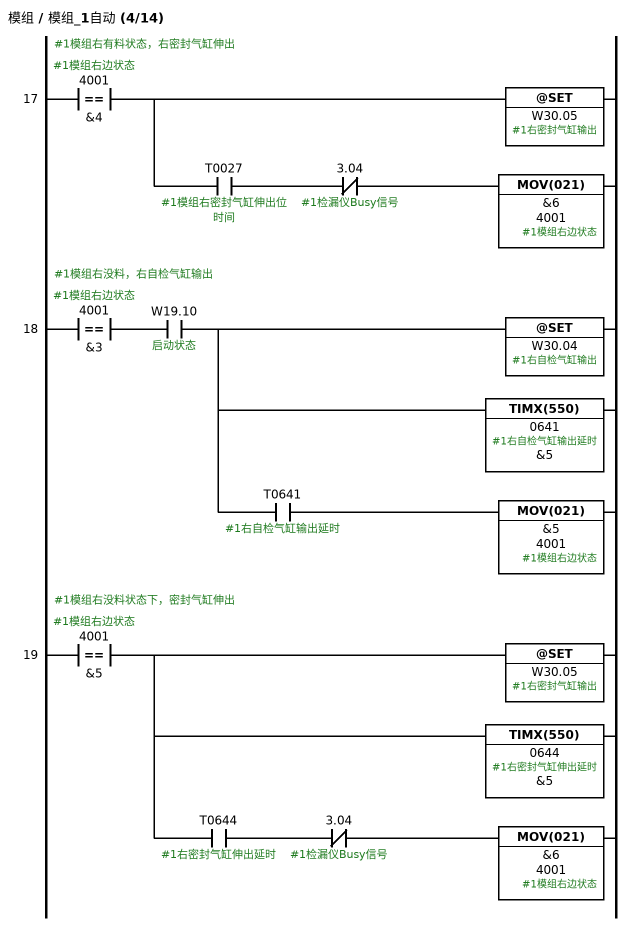
; [picture p209: 模组 / 模组_1自动, rungs 17-19]
; rung 17: #1模组右有料状态，右密封气缸伸出
LD=(300) 4001 &4  ; #1模组右边状态
@SET W30.05  ; #1右密封气缸输出
AND T0027  ; #1模组右密封气缸伸出位时间
ANDNOT 3.04  ; #1检漏仪Busy信号
MOV(021) &6 4001  ; #1模组右边状态
; rung 18: #1模组右没料，右自检气缸输出
LD=(300) 4001 &3  ; #1模组右边状态
AND W19.10  ; 启动状态
@SET W30.04  ; #1右自检气缸输出
TIMX(550) 0641 &5  ; #1右自检气缸输出延时
AND T0641  ; #1右自检气缸输出延时
MOV(021) &5 4001  ; #1模组右边状态
; rung 19: #1模组右没料状态下，密封气缸伸出
LD=(300) 4001 &5  ; #1模组右边状态
@SET W30.05  ; #1右密封气缸输出
TIMX(550) 0644 &5  ; #1右密封气缸伸出延时
AND T0644  ; #1右密封气缸伸出延时
ANDNOT 3.04  ; #1检漏仪Busy信号
MOV(021) &6 4001  ; #1模组右边状态

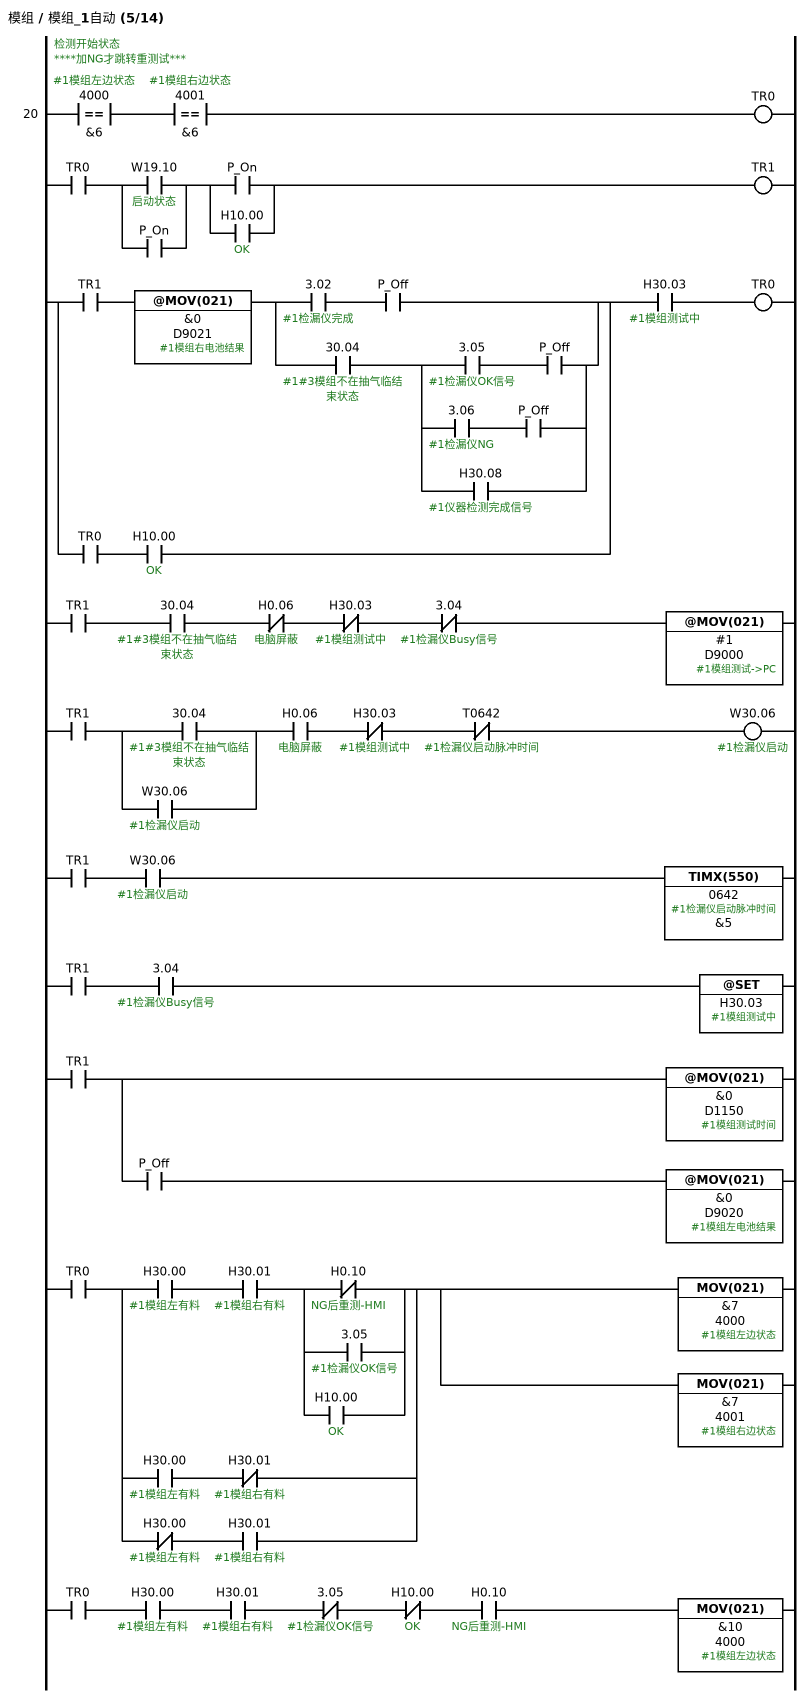
; rung 20: 检测开始状态 / ****加NG才跳转重测试***
LD=(300) 4000 &6  ; #1模组左边状态
AND=(300) 4001 &6  ; #1模组右边状态
OUT TR0
LD W19.10  ; 启动状态
OR P_On
ANDLD
LD P_On
OR H10.00  ; OK
ANDLD
OUT TR1
AND 30.04  ; #1#3模组不在抽气临结束状态  // 2018/5/28hy修改 所有模组不在抽气临结束状态下，下一模组才能启动(防抽气NG)
ANDNOT H0.06  ; 电脑屏蔽
ANDNOT H30.03  ; #1模组测试中
ANDNOT 3.04  ; #1检漏仪Busy信号
@MOV(021) #1 D9000  ; #1模组测试->PC
LD TR1
LD 30.04  ; #1#3模组不在抽气临结束状态  // 2018/5/28hy修改 所有模组不在抽气临结束状态下，下一模组才能启动(防抽气NG)
OR W30.06  ; #1检漏仪启动
ANDLD
AND H0.06  ; 电脑屏蔽
ANDNOT H30.03  ; #1模组测试中
ANDNOT T0642  ; #1检漏仪启动脉冲时间
OUT W30.06  ; #1检漏仪启动
LD TR1
AND W30.06  ; #1检漏仪启动
TIMX(550) 0642 &5  ; #1检漏仪启动脉冲时间
LD TR1
AND 3.04  ; #1检漏仪Busy信号
@SET H30.03  ; #1模组测试中
LD TR1
@MOV(021) &0 D1150  ; #1模组测试时间
AND P_Off
@MOV(021) &0 D9020  ; #1模组左电池结果
LD TR1
@MOV(021) &0 D9021  ; #1模组右电池结果
LD 3.02  ; #1检漏仪完成
AND P_Off
LD 30.04  ; #1#3模组不在抽气临结束状态  // 2018/5/29hy修改,所有模组不在临抽气结束状态下，测试模组测试完成后，给出停止测试信号
LD 3.05  ; #1检漏仪OK信号
AND P_Off
LD 3.06  ; #1检漏仪NG
AND P_Off
ORLD
OR H30.08  ; #1仪器检测完成信号
ANDLD
ORLD
ANDLD
LD TR0
AND H10.00  ; OK
ORLD
AND H30.03  ; #1模组测试中
OUT TR0
LD H30.00  ; #1模组左有料
AND H30.01  ; #1模组右有料
LDNOT H0.10  ; NG后重测-HMI
OR 3.05  ; #1检漏仪OK信号
OR H10.00  ; OK
ANDLD
LD H30.00  ; #1模组左有料
ANDNOT H30.01  ; #1模组右有料
ORLD
LDNOT H30.00  ; #1模组左有料
AND H30.01  ; #1模组右有料
ORLD
ANDLD
MOV(021) &7 4000  ; #1模组左边状态
MOV(021) &7 4001  ; #1模组右边状态
LD TR0
AND H30.00  ; #1模组左有料
AND H30.01  ; #1模组右有料
ANDNOT 3.05  ; #1检漏仪OK信号
ANDNOT H10.00  ; OK
AND H0.10  ; NG后重测-HMI
MOV(021) &10 4000  ; #1模组左边状态

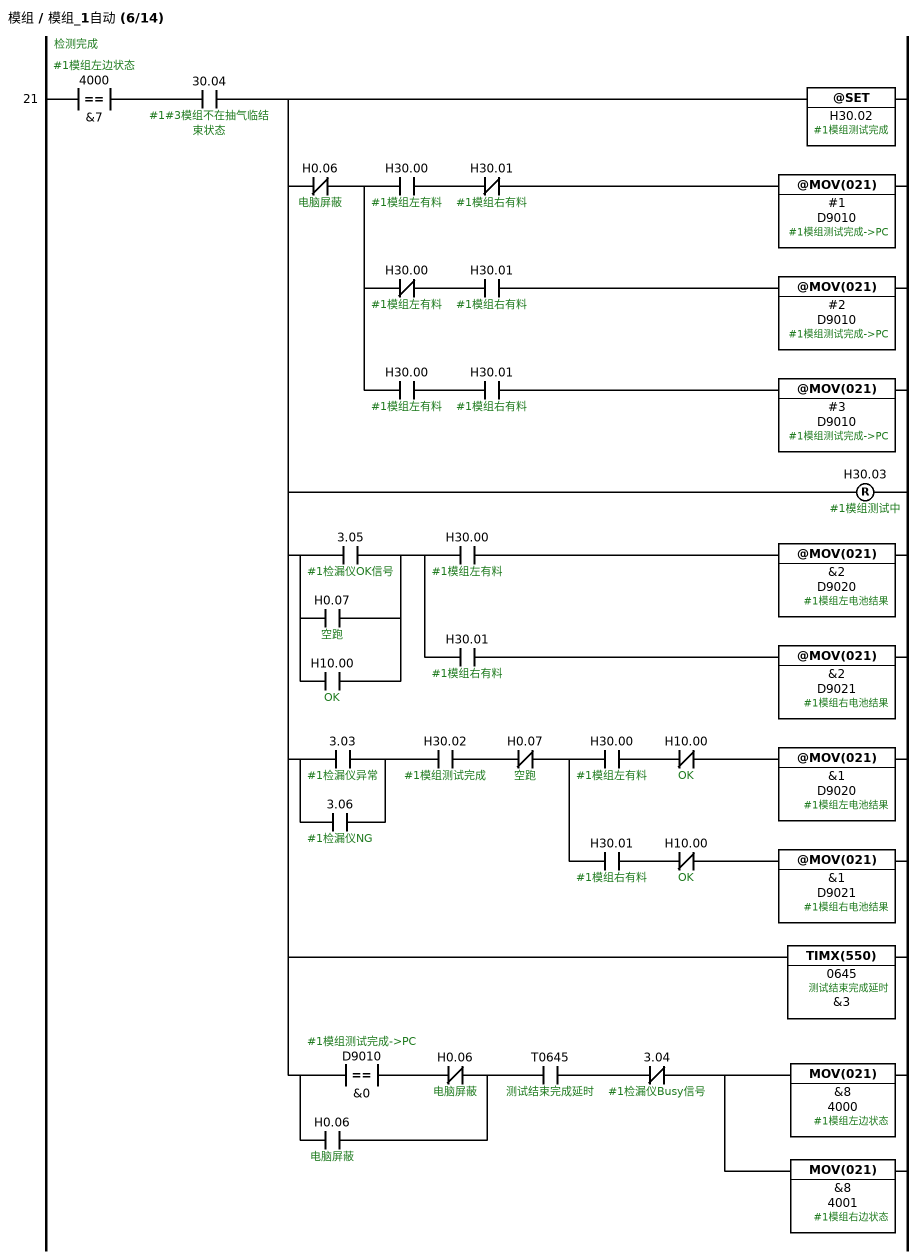
; rung 21: 检测完成
LD=(300) 4000 &7  ; #1模组左边状态
AND 30.04  ; #1#3模组不在抽气临结束状态
OUT TR0
@SET H30.02  ; #1模组测试完成
ANDNOT H0.06  ; 电脑屏蔽
OUT TR1
AND H30.00  ; #1模组左有料
ANDNOT H30.01  ; #1模组右有料
@MOV(021) #1 D9010  ; #1模组测试完成->PC
LD TR1
ANDNOT H30.00  ; #1模组左有料
AND H30.01  ; #1模组右有料
@MOV(021) #2 D9010  ; #1模组测试完成->PC
LD TR1
AND H30.00  ; #1模组左有料
AND H30.01  ; #1模组右有料
@MOV(021) #3 D9010  ; #1模组测试完成->PC
LD TR0
RSET H30.03  ; #1模组测试中
LD 3.05  ; #1检漏仪OK信号
OR H0.07  ; 空跑
OR H10.00  ; OK
ANDLD
OUT TR1
AND H30.00  ; #1模组左有料
@MOV(021) &2 D9020  ; #1模组左电池结果
LD TR1
AND H30.01  ; #1模组右有料
@MOV(021) &2 D9021  ; #1模组右电池结果
LD TR0
LD 3.03  ; #1检漏仪异常
OR 3.06  ; #1检漏仪NG
ANDLD
AND H30.02  ; #1模组测试完成
ANDNOT H0.07  ; 空跑
OUT TR1
AND H30.00  ; #1模组左有料
ANDNOT H10.00  ; OK
@MOV(021) &1 D9020  ; #1模组左电池结果
LD TR1
AND H30.01  ; #1模组右有料
ANDNOT H10.00  ; OK
@MOV(021) &1 D9021  ; #1模组右电池结果
LD TR0
TIMX(550) 0645 &3  ; 测试结束完成延时
LD=(300) D9010 &0  ; #1模组测试完成->PC
ANDNOT H0.06  ; 电脑屏蔽
OR H0.06  ; 电脑屏蔽
ANDLD
AND T0645  ; 测试结束完成延时
ANDNOT 3.04  ; #1检漏仪Busy信号
MOV(021) &8 4000  ; #1模组左边状态
MOV(021) &8 4001  ; #1模组右边状态

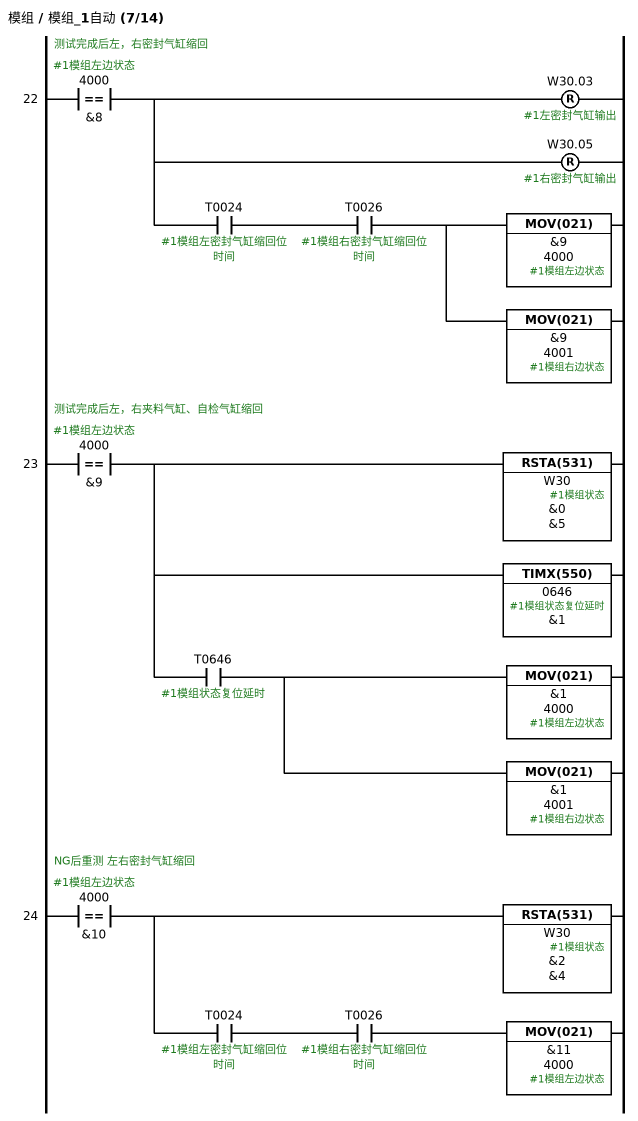
; rung 22: 测试完成后左，右密封气缸缩回
LD=(300) 4000 &8  ; #1模组左边状态
RSET W30.03  ; #1左密封气缸输出
RSET W30.05  ; #1右密封气缸输出
AND T0024  ; #1模组左密封气缸缩回位时间
AND T0026  ; #1模组右密封气缸缩回位时间
MOV(021) &9 4000  ; #1模组左边状态
MOV(021) &9 4001  ; #1模组右边状态
; rung 23: 测试完成后左，右夹料气缸、自检气缸缩回
LD=(300) 4000 &9  ; #1模组左边状态
RSTA(531) W30 &0 &5  ; #1模组状态
TIMX(550) 0646 &1  ; #1模组状态复位延时
AND T0646  ; #1模组状态复位延时
MOV(021) &1 4000  ; #1模组左边状态
MOV(021) &1 4001  ; #1模组右边状态
; rung 24: NG后重测 左右密封气缸缩回
LD=(300) 4000 &10  ; #1模组左边状态
RSTA(531) W30 &2 &4  ; #1模组状态
AND T0024  ; #1模组左密封气缸缩回位时间
AND T0026  ; #1模组右密封气缸缩回位时间
MOV(021) &11 4000  ; #1模组左边状态

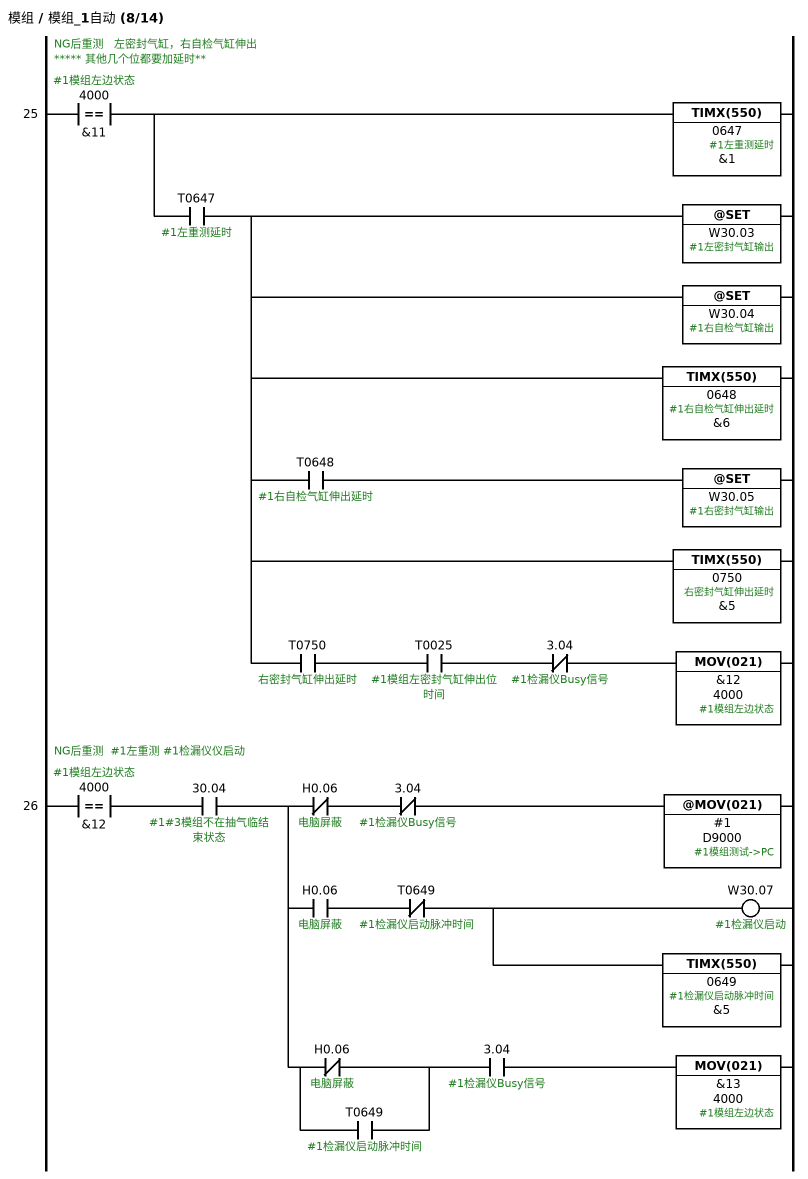
; rung 25: NG后重测   左密封气缸，右自检气缸伸出 / ***** 其他几个位都要加延时**
LD=(300) 4000 &11  ; #1模组左边状态
TIMX(550) 0647 &1  ; #1左重测延时
AND T0647  ; #1左重测延时
OUT TR0
@SET W30.03  ; #1左密封气缸输出
@SET W30.04  ; #1右自检气缸输出
TIMX(550) 0648 &6  ; #1右自检气缸伸出延时
AND T0648  ; #1右自检气缸伸出延时
@SET W30.05  ; #1右密封气缸输出
LD TR0
TIMX(550) 0750 &5  ; 右密封气缸伸出延时
AND T0750  ; 右密封气缸伸出延时
AND T0025  ; #1模组左密封气缸伸出位时间
ANDNOT 3.04  ; #1检漏仪Busy信号
MOV(021) &12 4000  ; #1模组左边状态
; rung 26: NG后重测  #1左重测 #1检漏仪仪启动
LD=(300) 4000 &12  ; #1模组左边状态
AND 30.04  ; #1#3模组不在抽气临结束状态  // 2018/5/28hy修改 所有模组不在抽气临结束状态下，下一模组才能启动(防抽气NG)
OUT TR0
ANDNOT H0.06  ; 电脑屏蔽
ANDNOT 3.04  ; #1检漏仪Busy信号
@MOV(021) #1 D9000  ; #1模组测试->PC
LD TR0
AND H0.06  ; 电脑屏蔽
ANDNOT T0649  ; #1检漏仪启动脉冲时间
OUT W30.07  ; #1检漏仪启动
TIMX(550) 0649 &5  ; #1检漏仪启动脉冲时间
LD TR0
LDNOT H0.06  ; 电脑屏蔽
OR T0649  ; #1检漏仪启动脉冲时间
ANDLD
AND 3.04  ; #1检漏仪Busy信号
MOV(021) &13 4000  ; #1模组左边状态

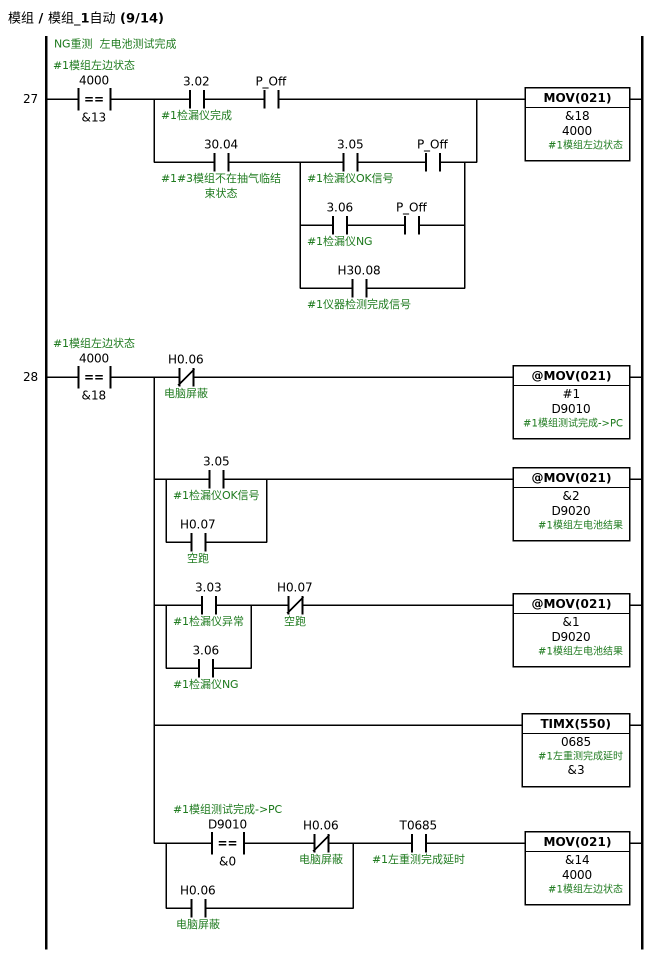
; rung 27: NG重测  左电池测试完成
LD=(300) 4000 &13  ; #1模组左边状态
LD 3.02  ; #1检漏仪完成
AND P_Off
LD 30.04  ; #1#3模组不在抽气临结束状态  // 2018/5/29hy修改,所有模组不在临抽气结束状态下，测试模组测试完成后，给出停止测试信号
LD 3.05  ; #1检漏仪OK信号
AND P_Off
LD 3.06  ; #1检漏仪NG
AND P_Off
ORLD
OR H30.08  ; #1仪器检测完成信号
ANDLD
ORLD
ANDLD
MOV(021) &18 4000  ; #1模组左边状态
; rung 28
LD=(300) 4000 &18  ; #1模组左边状态
OUT TR0
ANDNOT H0.06  ; 电脑屏蔽
@MOV(021) #1 D9010  ; #1模组测试完成->PC
LD TR0
LD 3.05  ; #1检漏仪OK信号
OR H0.07  ; 空跑
ANDLD
@MOV(021) &2 D9020  ; #1模组左电池结果
LD TR0
LD 3.03  ; #1检漏仪异常
OR 3.06  ; #1检漏仪NG
ANDLD
ANDNOT H0.07  ; 空跑
@MOV(021) &1 D9020  ; #1模组左电池结果
LD TR0
TIMX(550) 0685 &3  ; #1左重测完成延时
LD=(300) D9010 &0  ; #1模组测试完成->PC
ANDNOT H0.06  ; 电脑屏蔽
OR H0.06  ; 电脑屏蔽
ANDLD
AND T0685  ; #1左重测完成延时
MOV(021) &14 4000  ; #1模组左边状态

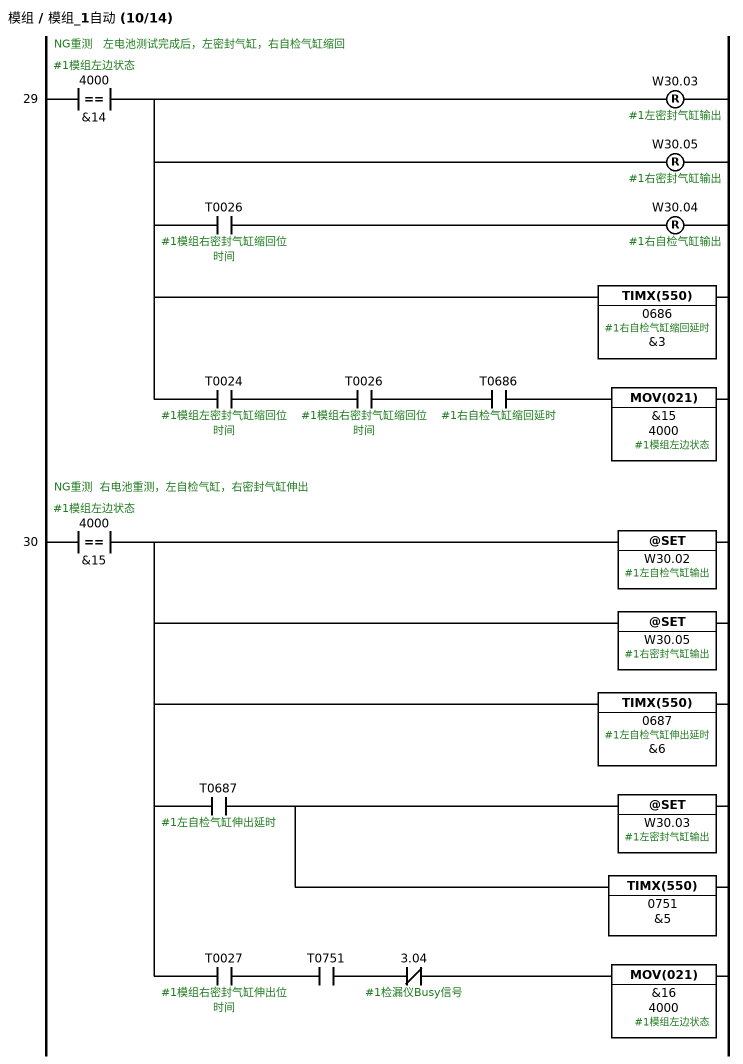
; rung 29: NG重测   左电池测试完成后，左密封气缸，右自检气缸缩回
LD=(300) 4000 &14  ; #1模组左边状态
OUT TR0
RSET W30.03  ; #1左密封气缸输出
RSET W30.05  ; #1右密封气缸输出
AND T0026  ; #1模组右密封气缸缩回位时间
RSET W30.04  ; #1右自检气缸输出
LD TR0
TIMX(550) 0686 &3  ; #1右自检气缸缩回延时
AND T0024  ; #1模组左密封气缸缩回位时间
AND T0026  ; #1模组右密封气缸缩回位时间
AND T0686  ; #1右自检气缸缩回延时
MOV(021) &15 4000  ; #1模组左边状态
; rung 30: NG重测  右电池重测，左自检气缸，右密封气缸伸出
LD=(300) 4000 &15  ; #1模组左边状态
OUT TR0
@SET W30.02  ; #1左自检气缸输出
@SET W30.05  ; #1右密封气缸输出
TIMX(550) 0687 &6  ; #1左自检气缸伸出延时
AND T0687  ; #1左自检气缸伸出延时
@SET W30.03  ; #1左密封气缸输出
TIMX(550) 0751 &5
LD TR0
AND T0027  ; #1模组右密封气缸伸出位时间
AND T0751
ANDNOT 3.04  ; #1检漏仪Busy信号
MOV(021) &16 4000  ; #1模组左边状态

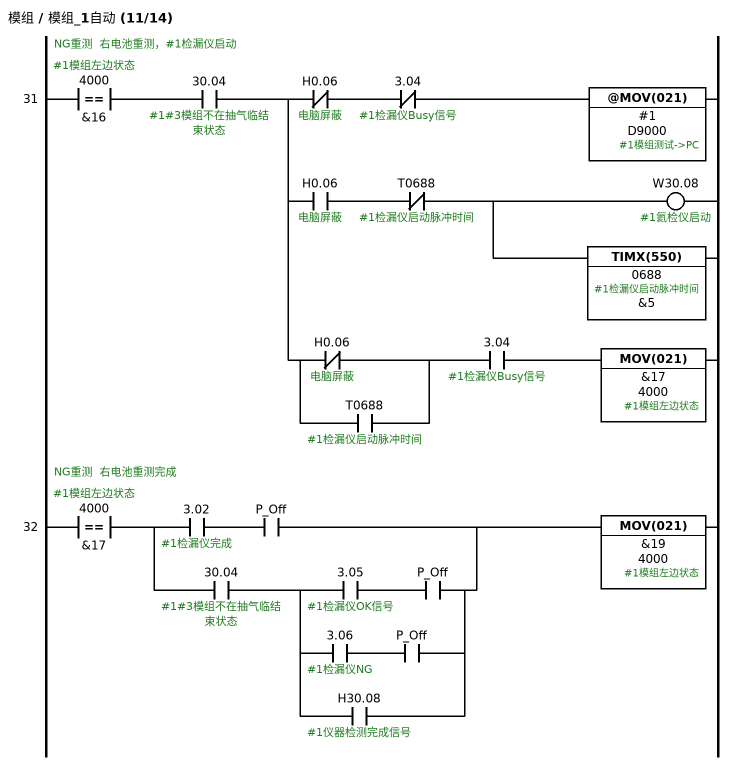
; rung 31: NG重测  右电池重测，#1检漏仪启动
LD=(300) 4000 &16  ; #1模组左边状态
AND 30.04  ; #1#3模组不在抽气临结束状态  // 2018/5/28hy修改 所有模组不在抽气临结束状态下，下一模组才能启动(防抽气NG)
OUT TR0
ANDNOT H0.06  ; 电脑屏蔽
ANDNOT 3.04  ; #1检漏仪Busy信号
@MOV(021) #1 D9000  ; #1模组测试->PC
LD TR0
AND H0.06  ; 电脑屏蔽
ANDNOT T0688  ; #1检漏仪启动脉冲时间
OUT W30.08  ; #1氦检仪启动
TIMX(550) 0688 &5  ; #1检漏仪启动脉冲时间
LD TR0
LDNOT H0.06  ; 电脑屏蔽
OR T0688  ; #1检漏仪启动脉冲时间
ANDLD
AND 3.04  ; #1检漏仪Busy信号
MOV(021) &17 4000  ; #1模组左边状态
; rung 32: NG重测  右电池重测完成
LD=(300) 4000 &17  ; #1模组左边状态
LD 3.02  ; #1检漏仪完成
AND P_Off
LD 30.04  ; #1#3模组不在抽气临结束状态  // 2018/5/29hy修改,所有模组不在临抽气结束状态下，测试模组测试完成后，给出停止测试信号
LD 3.05  ; #1检漏仪OK信号
AND P_Off
LD 3.06  ; #1检漏仪NG
AND P_Off
ORLD
OR H30.08  ; #1仪器检测完成信号
ANDLD
ORLD
ANDLD
MOV(021) &19 4000  ; #1模组左边状态

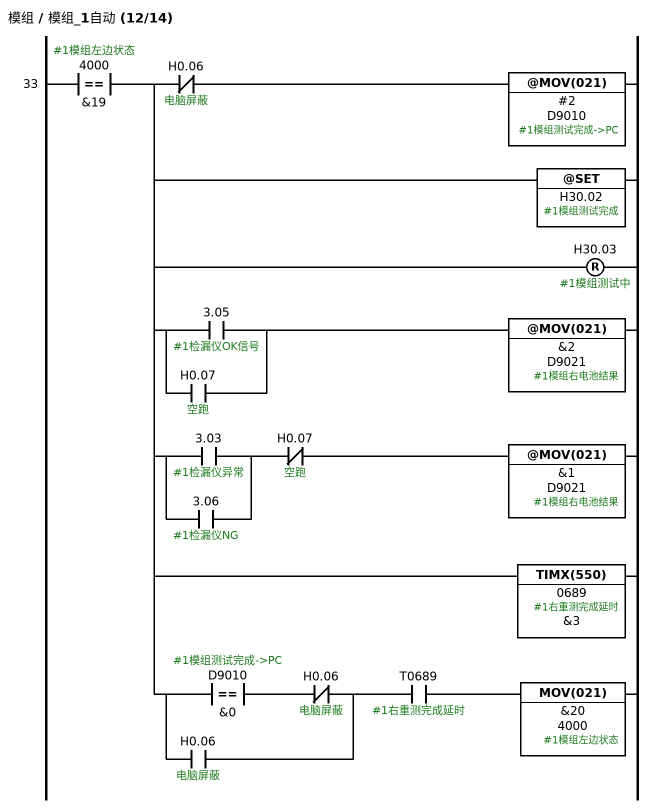
; rung 33
LD=(300) 4000 &19  ; #1模组左边状态
OUT TR0
ANDNOT H0.06  ; 电脑屏蔽
@MOV(021) #2 D9010  ; #1模组测试完成->PC
LD TR0
@SET H30.02  ; #1模组测试完成
RSET H30.03  ; #1模组测试中
LD 3.05  ; #1检漏仪OK信号
OR H0.07  ; 空跑
ANDLD
@MOV(021) &2 D9021  ; #1模组右电池结果
LD TR0
LD 3.03  ; #1检漏仪异常
OR 3.06  ; #1检漏仪NG
ANDLD
ANDNOT H0.07  ; 空跑
@MOV(021) &1 D9021  ; #1模组右电池结果
LD TR0
TIMX(550) 0689 &3  ; #1右重测完成延时
LD=(300) D9010 &0  ; #1模组测试完成->PC
ANDNOT H0.06  ; 电脑屏蔽
OR H0.06  ; 电脑屏蔽
ANDLD
AND T0689  ; #1右重测完成延时
MOV(021) &20 4000  ; #1模组左边状态

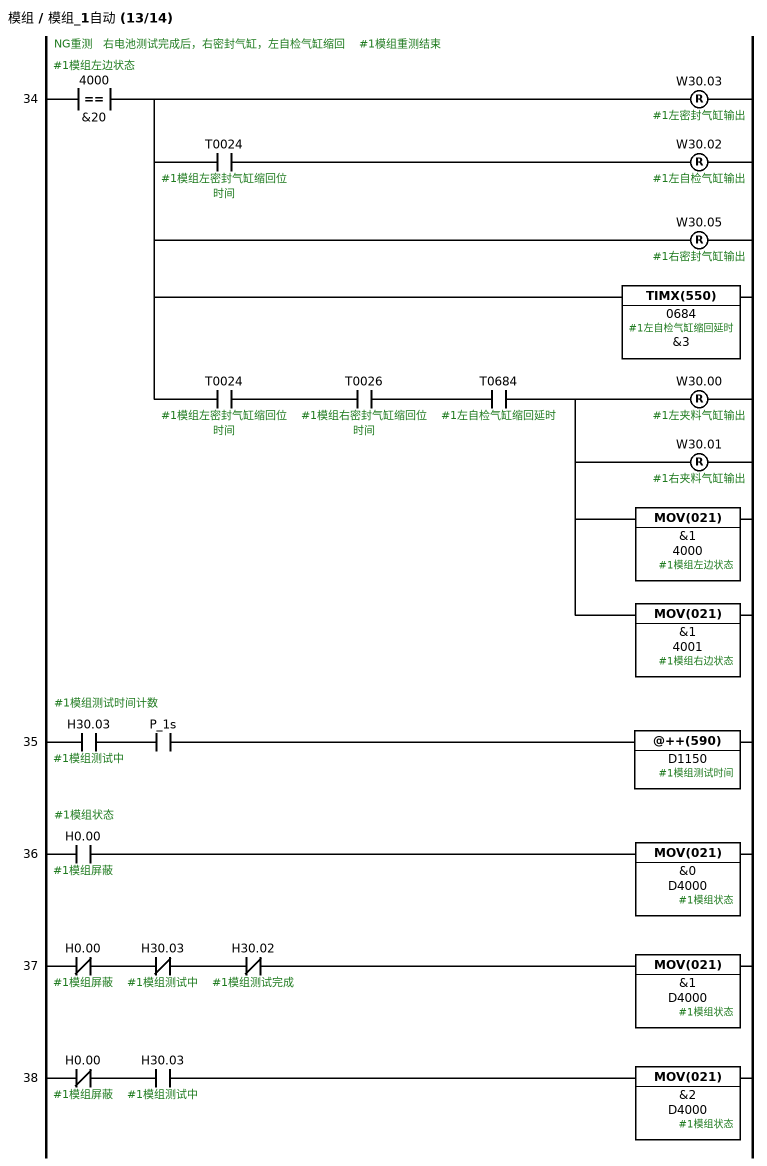
; rung 34: NG重测   右电池测试完成后，右密封气缸，左自检气缸缩回    #1模组重测结束
LD=(300) 4000 &20  ; #1模组左边状态
OUT TR0
RSET W30.03  ; #1左密封气缸输出
AND T0024  ; #1模组左密封气缸缩回位时间
RSET W30.02  ; #1左自检气缸输出
LD TR0
RSET W30.05  ; #1右密封气缸输出
TIMX(550) 0684 &3  ; #1左自检气缸缩回延时
AND T0024  ; #1模组左密封气缸缩回位时间
AND T0026  ; #1模组右密封气缸缩回位时间
AND T0684  ; #1左自检气缸缩回延时
RSET W30.00  ; #1左夹料气缸输出
RSET W30.01  ; #1右夹料气缸输出
MOV(021) &1 4000  ; #1模组左边状态
MOV(021) &1 4001  ; #1模组右边状态
; rung 35: #1模组测试时间计数
LD H30.03  ; #1模组测试中
AND P_1s
@++(590) D1150  ; #1模组测试时间
; rung 36: #1模组状态
LD H0.00  ; #1模组屏蔽
MOV(021) &0 D4000  ; #1模组状态
; rung 37
LDNOT H0.00  ; #1模组屏蔽
ANDNOT H30.03  ; #1模组测试中
ANDNOT H30.02  ; #1模组测试完成
MOV(021) &1 D4000  ; #1模组状态
; rung 38
LDNOT H0.00  ; #1模组屏蔽
AND H30.03  ; #1模组测试中
MOV(021) &2 D4000  ; #1模组状态

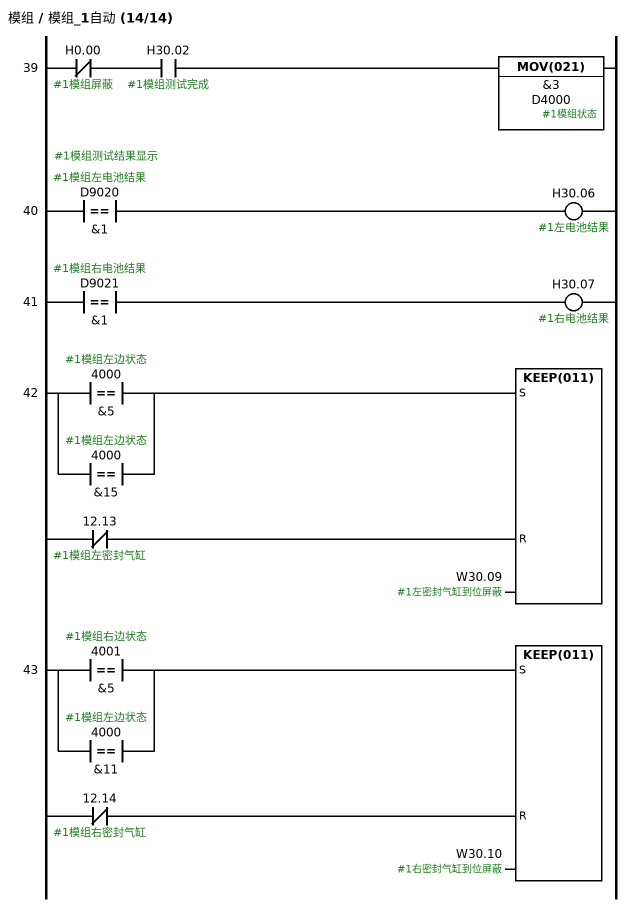
; rung 39
LDNOT H0.00  ; #1模组屏蔽
AND H30.02  ; #1模组测试完成
MOV(021) &3 D4000  ; #1模组状态
; rung 40: #1模组测试结果显示
LD=(300) D9020 &1  ; #1模组左电池结果
OUT H30.06  ; #1左电池结果
; rung 41
LD=(300) D9021 &1  ; #1模组右电池结果
OUT H30.07  ; #1右电池结果
; rung 42
LD=(300) 4000 &5  ; #1模组左边状态
OR=(300) 4000 &15  ; #1模组左边状态
LDNOT 12.13  ; #1模组左密封气缸
KEEP(011) W30.09  ; #1左密封气缸到位屏蔽
; rung 43
LD=(300) 4001 &5  ; #1模组右边状态
OR=(300) 4000 &11  ; #1模组左边状态
LDNOT 12.14  ; #1模组右密封气缸
KEEP(011) W30.10  ; #1右密封气缸到位屏蔽

### Section 模组_2自动

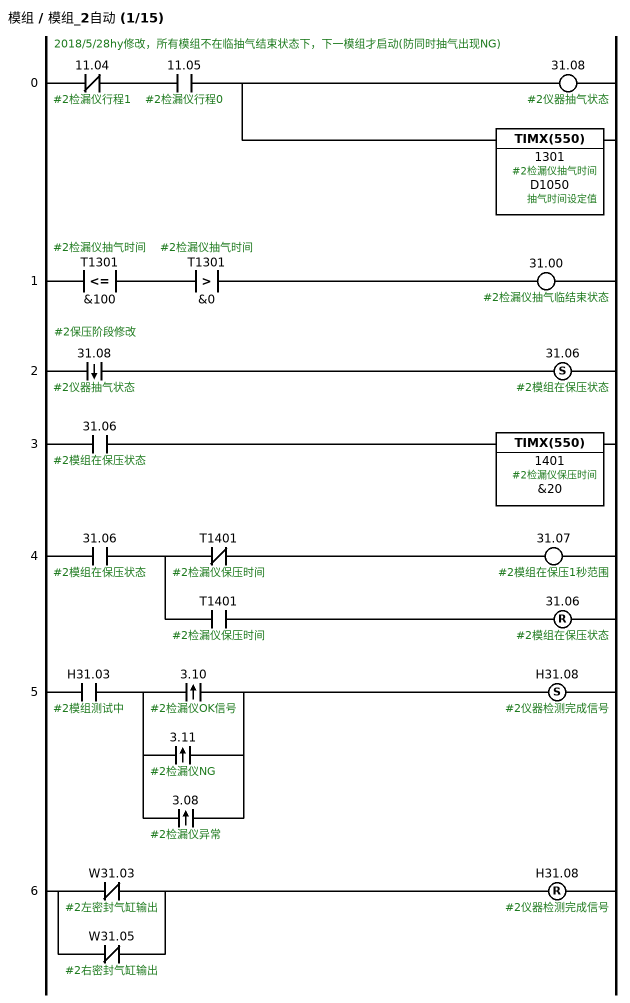
; rung 0: 2018/5/28hy修改，所有模组不在临抽气结束状态下，下一模组才启动(防同时抽气出现NG)
LDNOT 11.04  ; #2检漏仪行程1
AND 11.05  ; #2检漏仪行程0
OUT 31.08  ; #2仪器抽气状态
TIMX(550) 1301 D1050  ; 抽气时间设定值, #2检漏仪抽气时间
; rung 1
LD<=(315) T1301 &100  ; #2检漏仪抽气时间
AND>(320) T1301 &0  ; #2检漏仪抽气时间
OUT 31.00  ; #2检漏仪抽气临结束状态
; rung 2: #2保压阶段修改
%LD 31.08  ; #2仪器抽气状态
SET 31.06  ; #2模组在保压状态
; rung 3
LD 31.06  ; #2模组在保压状态
TIMX(550) 1401 &20  ; #2检漏仪保压时间
; rung 4
LD 31.06  ; #2模组在保压状态
OUT TR0
ANDNOT T1401  ; #2检漏仪保压时间
OUT 31.07  ; #2模组在保压1秒范围
LD TR0
AND T1401  ; #2检漏仪保压时间
RSET 31.06  ; #2模组在保压状态
; rung 5
LD H31.03  ; #2模组测试中
@LD 3.10  ; #2检漏仪OK信号
@OR 3.11  ; #2检漏仪NG
@OR 3.08  ; #2检漏仪异常
ANDLD
SET H31.08  ; #2仪器检测完成信号
; rung 6
LDNOT W31.03  ; #2左密封气缸输出
ORNOT W31.05  ; #2右密封气缸输出
RSET H31.08  ; #2仪器检测完成信号

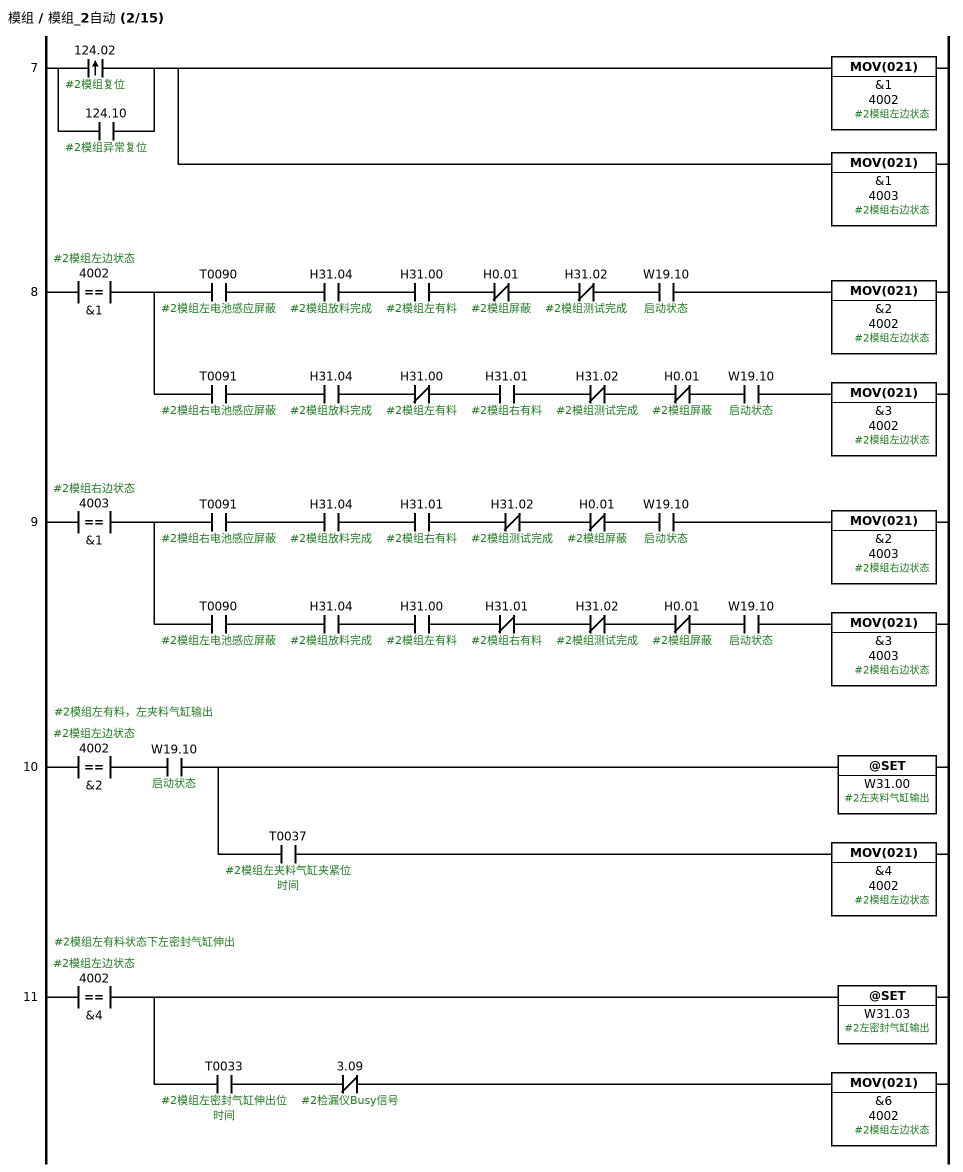
; rung 7
@LD 124.02  ; #2模组复位
OR 124.10  ; #2模组异常复位
MOV(021) &1 4002  ; #2模组左边状态
MOV(021) &1 4003  ; #2模组右边状态
; rung 8
LD=(300) 4002 &1  ; #2模组左边状态
OUT TR0
AND T0090  ; #2模组左电池感应屏蔽
AND H31.04  ; #2模组放料完成
AND H31.00  ; #2模组左有料
ANDNOT H0.01  ; #2模组屏蔽
ANDNOT H31.02  ; #2模组测试完成
AND W19.10  ; 启动状态
MOV(021) &2 4002  ; #2模组左边状态
LD TR0
AND T0091  ; #2模组右电池感应屏蔽
AND H31.04  ; #2模组放料完成
ANDNOT H31.00  ; #2模组左有料
AND H31.01  ; #2模组右有料
ANDNOT H31.02  ; #2模组测试完成
ANDNOT H0.01  ; #2模组屏蔽
AND W19.10  ; 启动状态
MOV(021) &3 4002  ; #2模组左边状态
; rung 9
LD=(300) 4003 &1  ; #2模组右边状态
OUT TR0
AND T0091  ; #2模组右电池感应屏蔽
AND H31.04  ; #2模组放料完成
AND H31.01  ; #2模组右有料
ANDNOT H31.02  ; #2模组测试完成
ANDNOT H0.01  ; #2模组屏蔽
AND W19.10  ; 启动状态
MOV(021) &2 4003  ; #2模组右边状态
LD TR0
AND T0090  ; #2模组左电池感应屏蔽
AND H31.04  ; #2模组放料完成
AND H31.00  ; #2模组左有料
ANDNOT H31.01  ; #2模组右有料
ANDNOT H31.02  ; #2模组测试完成
ANDNOT H0.01  ; #2模组屏蔽
AND W19.10  ; 启动状态
MOV(021) &3 4003  ; #2模组右边状态
; rung 10: #2模组左有料，左夹料气缸输出
LD=(300) 4002 &2  ; #2模组左边状态
AND W19.10  ; 启动状态
@SET W31.00  ; #2左夹料气缸输出
AND T0037  ; #2模组左夹料气缸夹紧位时间
MOV(021) &4 4002  ; #2模组左边状态
; rung 11: #2模组左有料状态下左密封气缸伸出
LD=(300) 4002 &4  ; #2模组左边状态
@SET W31.03  ; #2左密封气缸输出
AND T0033  ; #2模组左密封气缸伸出位时间
ANDNOT 3.09  ; #2检漏仪Busy信号
MOV(021) &6 4002  ; #2模组左边状态

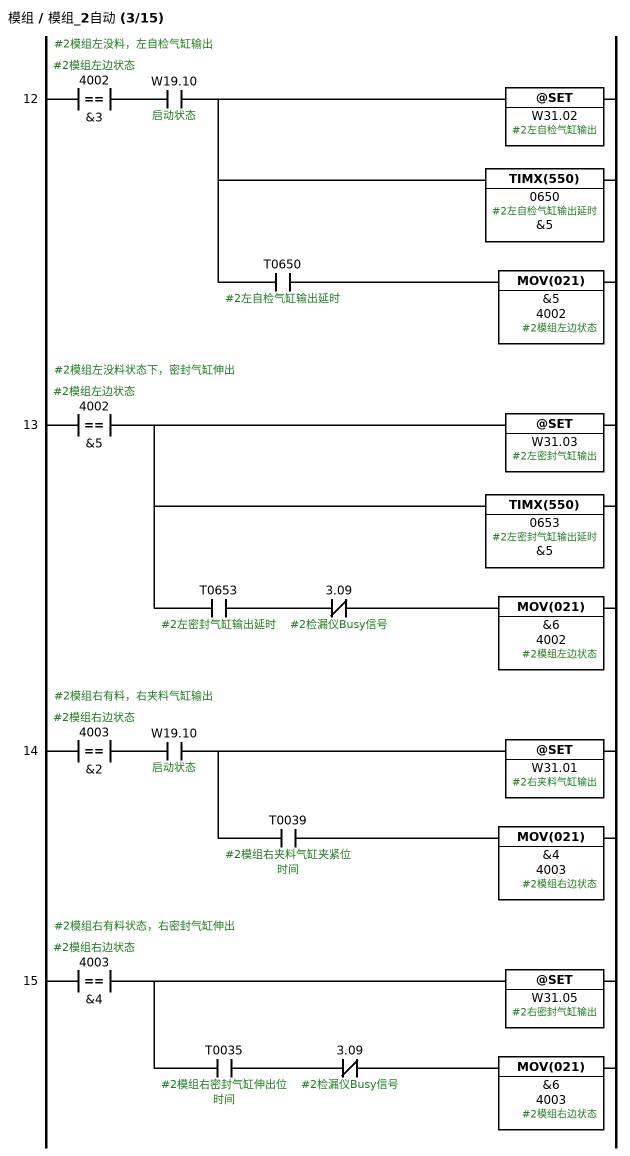
; rung 12: #2模组左没料，左自检气缸输出
LD=(300) 4002 &3  ; #2模组左边状态
AND W19.10  ; 启动状态
@SET W31.02  ; #2左自检气缸输出
TIMX(550) 0650 &5  ; #2左自检气缸输出延时
AND T0650  ; #2左自检气缸输出延时
MOV(021) &5 4002  ; #2模组左边状态
; rung 13: #2模组左没料状态下，密封气缸伸出
LD=(300) 4002 &5  ; #2模组左边状态
@SET W31.03  ; #2左密封气缸输出
TIMX(550) 0653 &5  ; #2左密封气缸输出延时
AND T0653  ; #2左密封气缸输出延时
ANDNOT 3.09  ; #2检漏仪Busy信号
MOV(021) &6 4002  ; #2模组左边状态
; rung 14: #2模组右有料，右夹料气缸输出
LD=(300) 4003 &2  ; #2模组右边状态
AND W19.10  ; 启动状态
@SET W31.01  ; #2右夹料气缸输出
AND T0039  ; #2模组右夹料气缸夹紧位时间
MOV(021) &4 4003  ; #2模组右边状态
; rung 15: #2模组右有料状态，右密封气缸伸出
LD=(300) 4003 &4  ; #2模组右边状态
@SET W31.05  ; #2右密封气缸输出
AND T0035  ; #2模组右密封气缸伸出位时间
ANDNOT 3.09  ; #2检漏仪Busy信号
MOV(021) &6 4003  ; #2模组右边状态

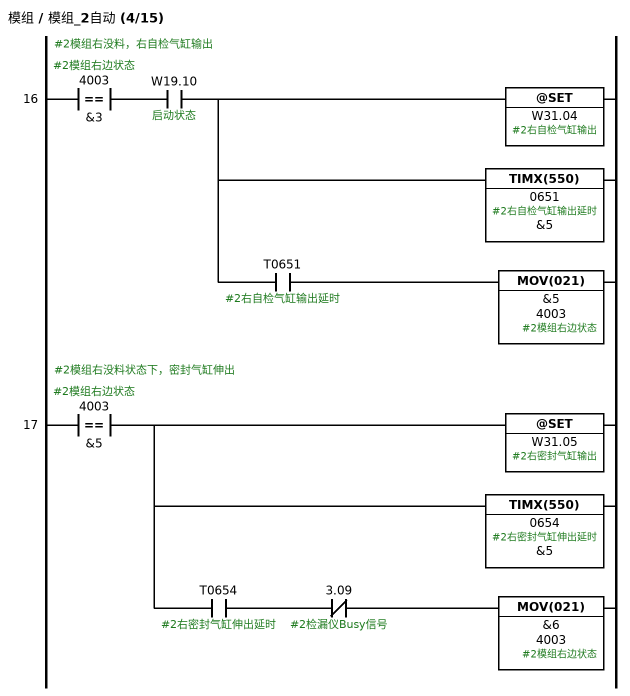
; rung 16: #2模组右没料，右自检气缸输出
LD=(300) 4003 &3  ; #2模组右边状态
AND W19.10  ; 启动状态
@SET W31.04  ; #2右自检气缸输出
TIMX(550) 0651 &5  ; #2右自检气缸输出延时
AND T0651  ; #2右自检气缸输出延时
MOV(021) &5 4003  ; #2模组右边状态
; rung 17: #2模组右没料状态下，密封气缸伸出
LD=(300) 4003 &5  ; #2模组右边状态
@SET W31.05  ; #2右密封气缸输出
TIMX(550) 0654 &5  ; #2右密封气缸伸出延时
AND T0654  ; #2右密封气缸伸出延时
ANDNOT 3.09  ; #2检漏仪Busy信号
MOV(021) &6 4003  ; #2模组右边状态

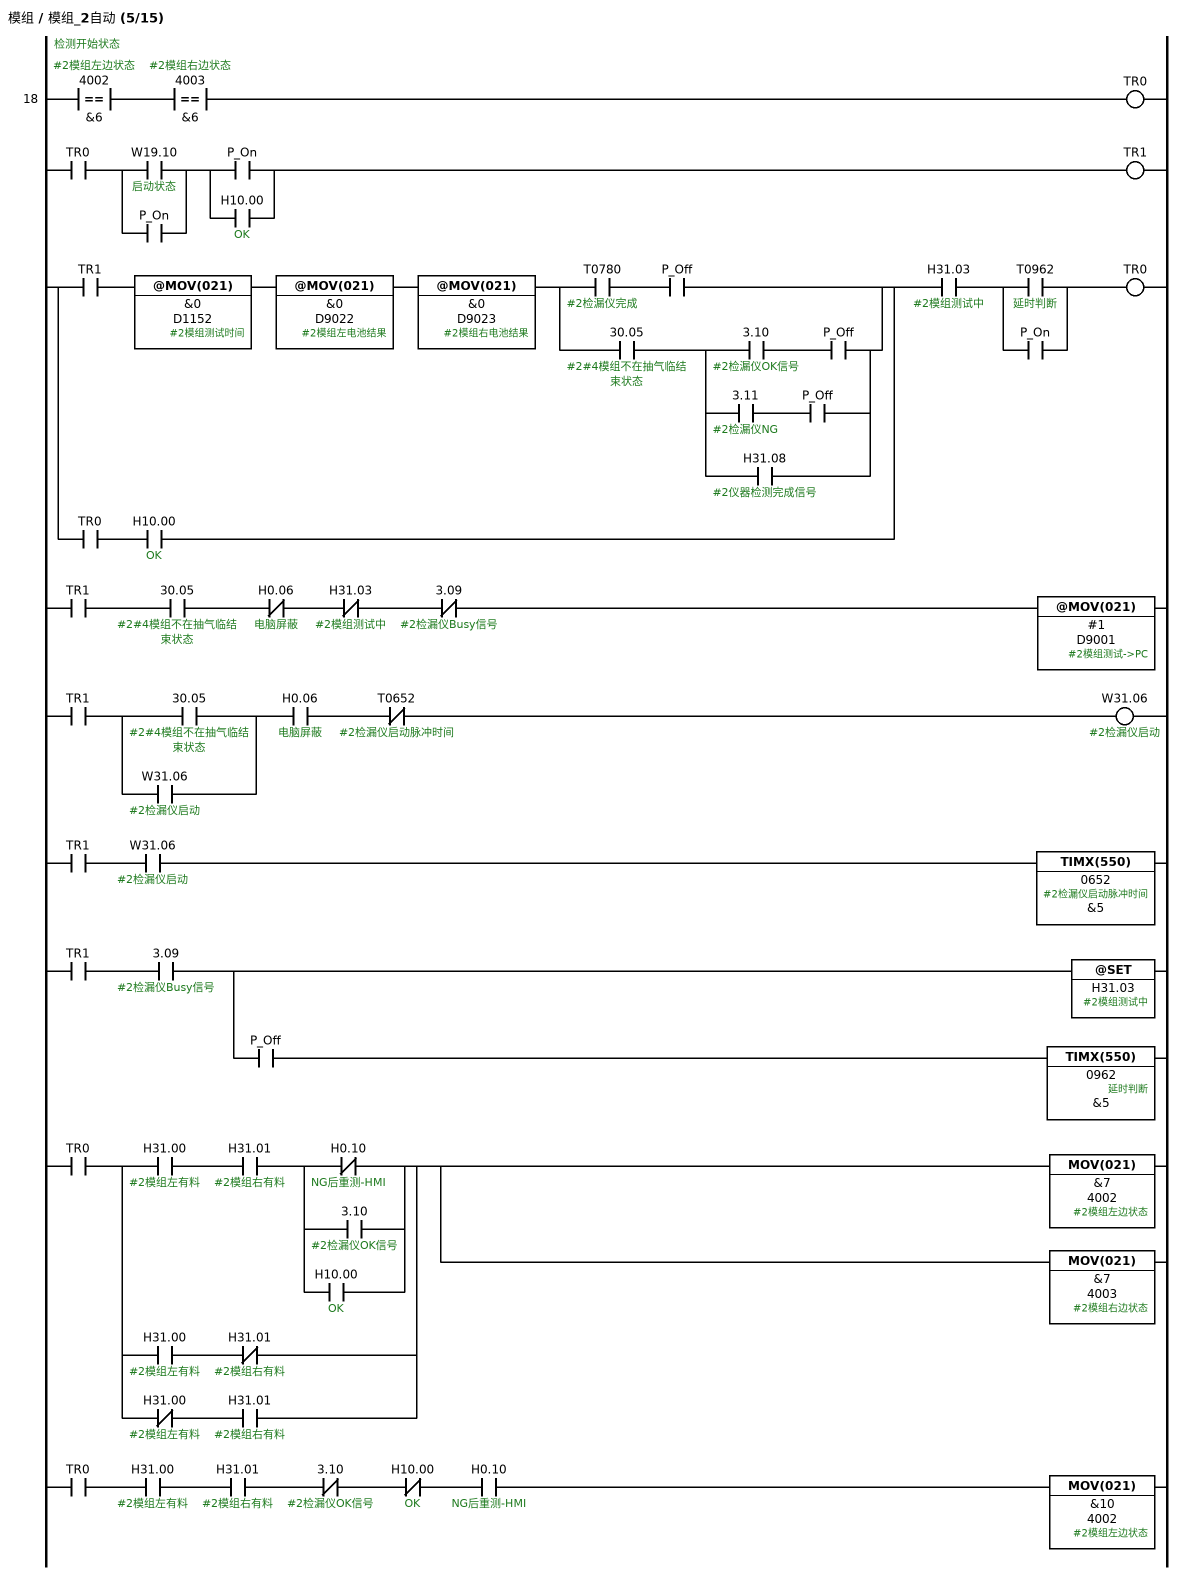
; rung 18: 检测开始状态
LD=(300) 4002 &6  ; #2模组左边状态
AND=(300) 4003 &6  ; #2模组右边状态
OUT TR0
LD W19.10  ; 启动状态
OR P_On
ANDLD
LD P_On  // 2018/5/28hy修改 所有模组不在抽气临结束状态下，下一模组才能启动(防抽气NG)
OR H10.00  ; OK
ANDLD
OUT TR1
AND 30.05  ; #2#4模组不在抽气临结束状态  // 2018/5/28hy修改 所有模组不在抽气临结束状态下，下一模组才能启动(防抽气NG)
ANDNOT H0.06  ; 电脑屏蔽
ANDNOT H31.03  ; #2模组测试中
ANDNOT 3.09  ; #2检漏仪Busy信号
@MOV(021) #1 D9001  ; #2模组测试->PC
LD TR1
LD 30.05  ; #2#4模组不在抽气临结束状态  // 2018/5/28hy修改 所有模组不在抽气临结束状态下，下一模组才能启动(防抽气NG)
OR W31.06  ; #2检漏仪启动
ANDLD
AND H0.06  ; 电脑屏蔽
ANDNOT T0652  ; #2检漏仪启动脉冲时间
OUT W31.06  ; #2检漏仪启动
LD TR1
AND W31.06  ; #2检漏仪启动
TIMX(550) 0652 &5  ; #2检漏仪启动脉冲时间
LD TR1
AND 3.09  ; #2检漏仪Busy信号
@SET H31.03  ; #2模组测试中
AND P_Off
TIMX(550) 0962 &5  ; 延时判断
LD TR1
@MOV(021) &0 D1152  ; #2模组测试时间
@MOV(021) &0 D9022  ; #2模组左电池结果
@MOV(021) &0 D9023  ; #2模组右电池结果
LD T0780  ; #2检漏仪完成
AND P_Off
LD 30.05  ; #2#4模组不在抽气临结束状态  // 2018/5/29hy修改,所有模组不在临抽气结束状态下，测试模组测试完成后，给出停止测试信号
LD 3.10  ; #2检漏仪OK信号
AND P_Off
LD 3.11  ; #2检漏仪NG
AND P_Off
ORLD
OR H31.08  ; #2仪器检测完成信号
ANDLD
ORLD
ANDLD
LD TR0
AND H10.00  ; OK
ORLD
AND H31.03  ; #2模组测试中
LD T0962  ; 延时判断
OR P_On
ANDLD
OUT TR0
LD H31.00  ; #2模组左有料
AND H31.01  ; #2模组右有料
LDNOT H0.10  ; NG后重测-HMI
OR 3.10  ; #2检漏仪OK信号
OR H10.00  ; OK
ANDLD
LD H31.00  ; #2模组左有料
ANDNOT H31.01  ; #2模组右有料
ORLD
LDNOT H31.00  ; #2模组左有料
AND H31.01  ; #2模组右有料
ORLD
ANDLD
MOV(021) &7 4002  ; #2模组左边状态
MOV(021) &7 4003  ; #2模组右边状态
LD TR0
AND H31.00  ; #2模组左有料
AND H31.01  ; #2模组右有料
ANDNOT 3.10  ; #2检漏仪OK信号
ANDNOT H10.00  ; OK
AND H0.10  ; NG后重测-HMI
MOV(021) &10 4002  ; #2模组左边状态

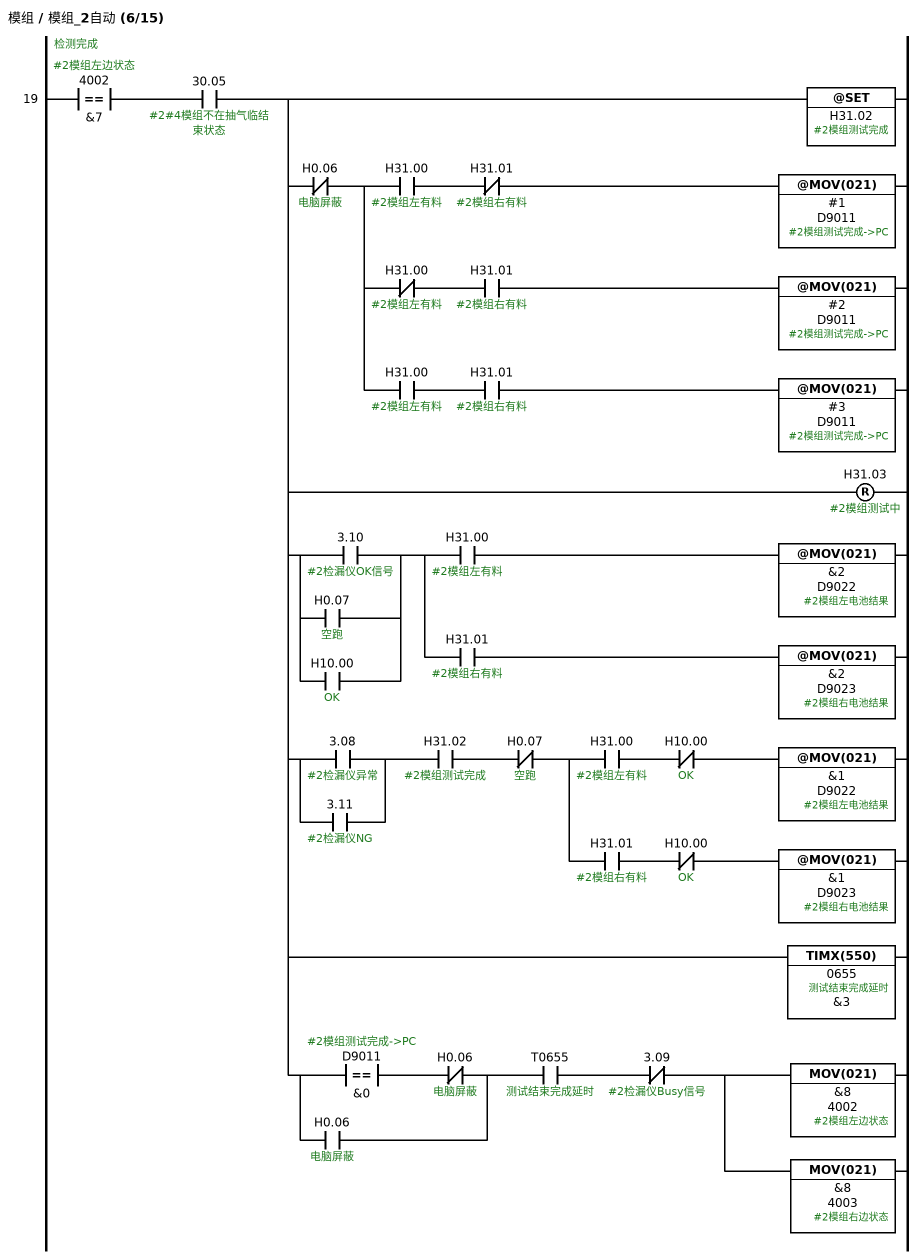
; rung 19: 检测完成
LD=(300) 4002 &7  ; #2模组左边状态
AND 30.05  ; #2#4模组不在抽气临结束状态
OUT TR0
@SET H31.02  ; #2模组测试完成
ANDNOT H0.06  ; 电脑屏蔽
OUT TR1
AND H31.00  ; #2模组左有料
ANDNOT H31.01  ; #2模组右有料
@MOV(021) #1 D9011  ; #2模组测试完成->PC
LD TR1
ANDNOT H31.00  ; #2模组左有料
AND H31.01  ; #2模组右有料
@MOV(021) #2 D9011  ; #2模组测试完成->PC
LD TR1
AND H31.00  ; #2模组左有料
AND H31.01  ; #2模组右有料
@MOV(021) #3 D9011  ; #2模组测试完成->PC
LD TR0
RSET H31.03  ; #2模组测试中
LD 3.10  ; #2检漏仪OK信号
OR H0.07  ; 空跑
OR H10.00  ; OK
ANDLD
OUT TR1
AND H31.00  ; #2模组左有料
@MOV(021) &2 D9022  ; #2模组左电池结果
LD TR1
AND H31.01  ; #2模组右有料
@MOV(021) &2 D9023  ; #2模组右电池结果
LD TR0
LD 3.08  ; #2检漏仪异常
OR 3.11  ; #2检漏仪NG
ANDLD
AND H31.02  ; #2模组测试完成
ANDNOT H0.07  ; 空跑
OUT TR1
AND H31.00  ; #2模组左有料
ANDNOT H10.00  ; OK
@MOV(021) &1 D9022  ; #2模组左电池结果
LD TR1
AND H31.01  ; #2模组右有料
ANDNOT H10.00  ; OK
@MOV(021) &1 D9023  ; #2模组右电池结果
LD TR0
TIMX(550) 0655 &3  ; 测试结束完成延时
LD=(300) D9011 &0  ; #2模组测试完成->PC
ANDNOT H0.06  ; 电脑屏蔽
OR H0.06  ; 电脑屏蔽
ANDLD
AND T0655  ; 测试结束完成延时
ANDNOT 3.09  ; #2检漏仪Busy信号
MOV(021) &8 4002  ; #2模组左边状态
MOV(021) &8 4003  ; #2模组右边状态

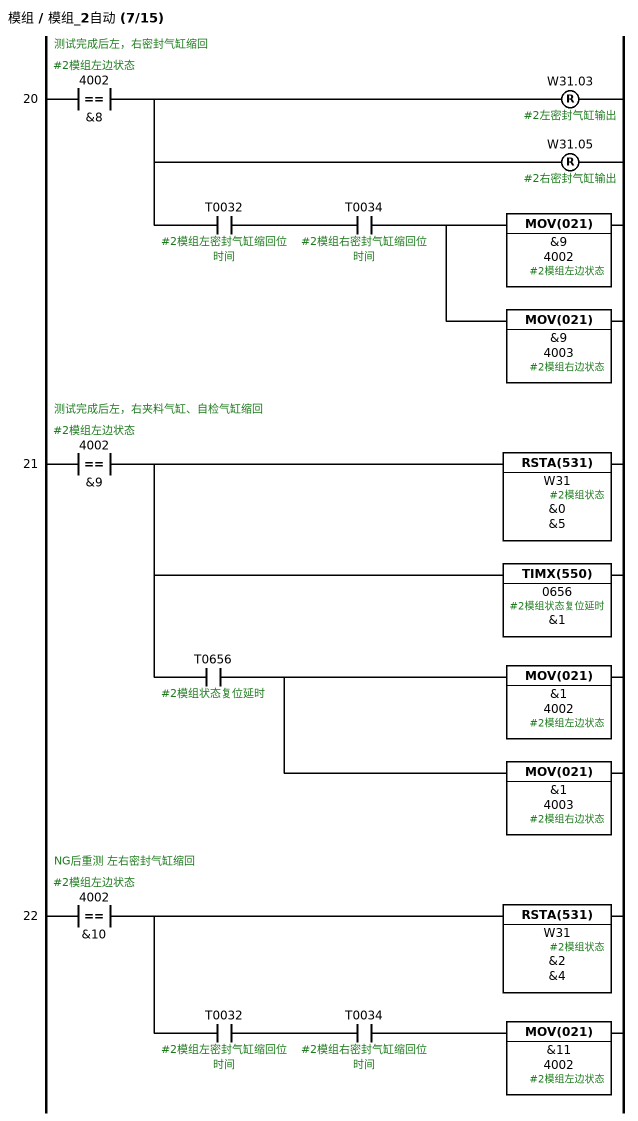
; rung 20: 测试完成后左，右密封气缸缩回
LD=(300) 4002 &8  ; #2模组左边状态
RSET W31.03  ; #2左密封气缸输出
RSET W31.05  ; #2右密封气缸输出
AND T0032  ; #2模组左密封气缸缩回位时间
AND T0034  ; #2模组右密封气缸缩回位时间
MOV(021) &9 4002  ; #2模组左边状态
MOV(021) &9 4003  ; #2模组右边状态
; rung 21: 测试完成后左，右夹料气缸、自检气缸缩回
LD=(300) 4002 &9  ; #2模组左边状态
RSTA(531) W31 &0 &5  ; #2模组状态
TIMX(550) 0656 &1  ; #2模组状态复位延时
AND T0656  ; #2模组状态复位延时
MOV(021) &1 4002  ; #2模组左边状态
MOV(021) &1 4003  ; #2模组右边状态
; rung 22: NG后重测 左右密封气缸缩回
LD=(300) 4002 &10  ; #2模组左边状态
RSTA(531) W31 &2 &4  ; #2模组状态
AND T0032  ; #2模组左密封气缸缩回位时间
AND T0034  ; #2模组右密封气缸缩回位时间
MOV(021) &11 4002  ; #2模组左边状态

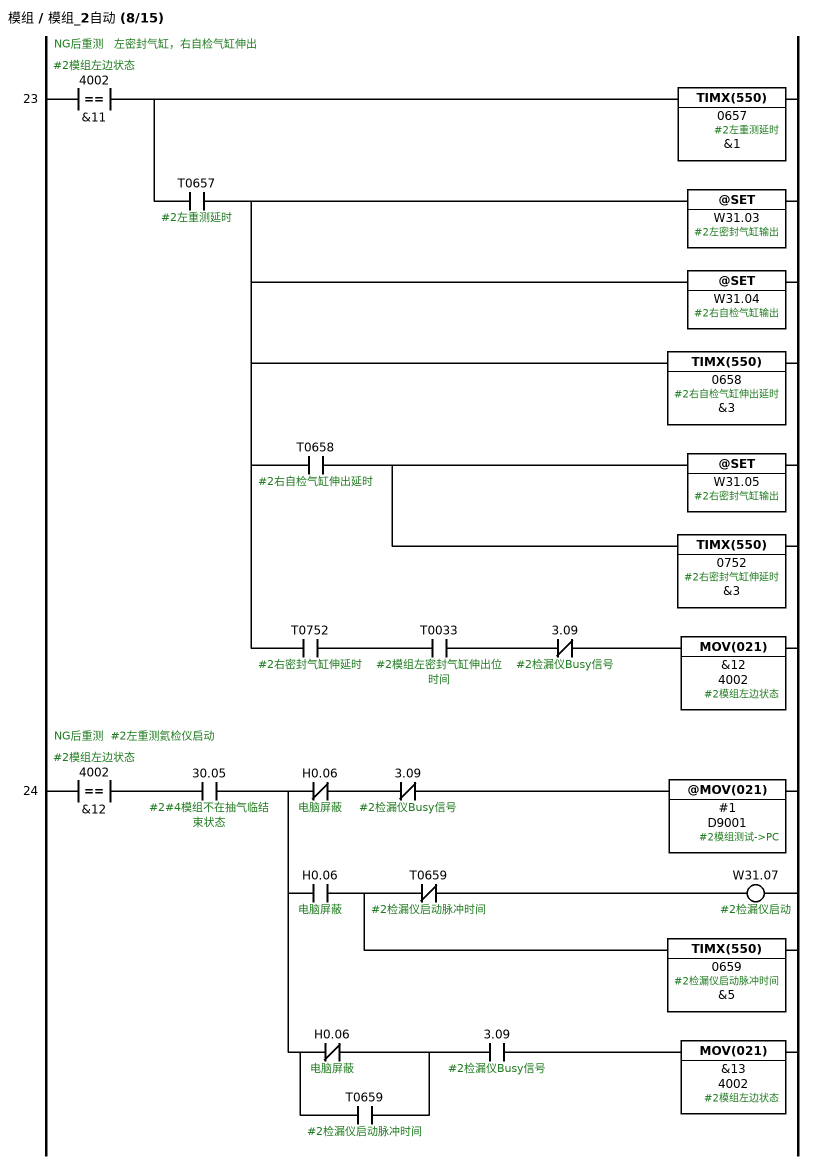
; rung 23: NG后重测   左密封气缸，右自检气缸伸出
LD=(300) 4002 &11  ; #2模组左边状态
TIMX(550) 0657 &1  ; #2左重测延时
AND T0657  ; #2左重测延时
OUT TR0
@SET W31.03  ; #2左密封气缸输出
@SET W31.04  ; #2右自检气缸输出
TIMX(550) 0658 &3  ; #2右自检气缸伸出延时
AND T0658  ; #2右自检气缸伸出延时
@SET W31.05  ; #2右密封气缸输出
TIMX(550) 0752 &3  ; #2右密封气缸伸延时
LD TR0
AND T0752  ; #2右密封气缸伸延时
AND T0033  ; #2模组左密封气缸伸出位时间
ANDNOT 3.09  ; #2检漏仪Busy信号
MOV(021) &12 4002  ; #2模组左边状态
; rung 24: NG后重测  #2左重测氦检仪启动
LD=(300) 4002 &12  ; #2模组左边状态
AND 30.05  ; #2#4模组不在抽气临结束状态  // 2018/5/28hy修改 所有模组不在抽气临结束状态下，下一模组才能启动(防抽气NG)
OUT TR0
ANDNOT H0.06  ; 电脑屏蔽
ANDNOT 3.09  ; #2检漏仪Busy信号
@MOV(021) #1 D9001  ; #2模组测试->PC
LD TR0
AND H0.06  ; 电脑屏蔽
OUT TR1
ANDNOT T0659  ; #2检漏仪启动脉冲时间
OUT W31.07  ; #2检漏仪启动
LD TR1
TIMX(550) 0659 &5  ; #2检漏仪启动脉冲时间
LD TR0
LDNOT H0.06  ; 电脑屏蔽
OR T0659  ; #2检漏仪启动脉冲时间
ANDLD
AND 3.09  ; #2检漏仪Busy信号
MOV(021) &13 4002  ; #2模组左边状态

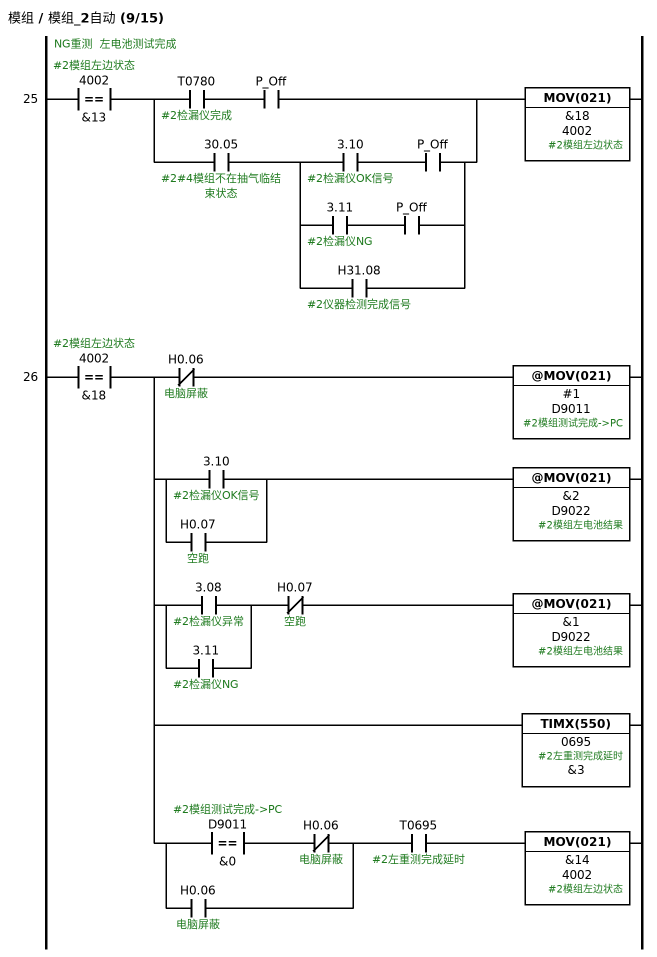
; rung 25: NG重测  左电池测试完成
LD=(300) 4002 &13  ; #2模组左边状态
LD T0780  ; #2检漏仪完成
AND P_Off
LD 30.05  ; #2#4模组不在抽气临结束状态  // 2018/5/29hy修改,所有模组不在临抽气结束状态下，测试模组测试完成后，给出停止测试信号
LD 3.10  ; #2检漏仪OK信号
AND P_Off
LD 3.11  ; #2检漏仪NG
AND P_Off
ORLD
OR H31.08  ; #2仪器检测完成信号
ANDLD
ORLD
ANDLD
MOV(021) &18 4002  ; #2模组左边状态
; rung 26
LD=(300) 4002 &18  ; #2模组左边状态
OUT TR0
ANDNOT H0.06  ; 电脑屏蔽
@MOV(021) #1 D9011  ; #2模组测试完成->PC
LD TR0
LD 3.10  ; #2检漏仪OK信号
OR H0.07  ; 空跑
ANDLD
@MOV(021) &2 D9022  ; #2模组左电池结果
LD TR0
LD 3.08  ; #2检漏仪异常
OR 3.11  ; #2检漏仪NG
ANDLD
ANDNOT H0.07  ; 空跑
@MOV(021) &1 D9022  ; #2模组左电池结果
LD TR0
TIMX(550) 0695 &3  ; #2左重测完成延时
LD=(300) D9011 &0  ; #2模组测试完成->PC
ANDNOT H0.06  ; 电脑屏蔽
OR H0.06  ; 电脑屏蔽
ANDLD
AND T0695  ; #2左重测完成延时
MOV(021) &14 4002  ; #2模组左边状态

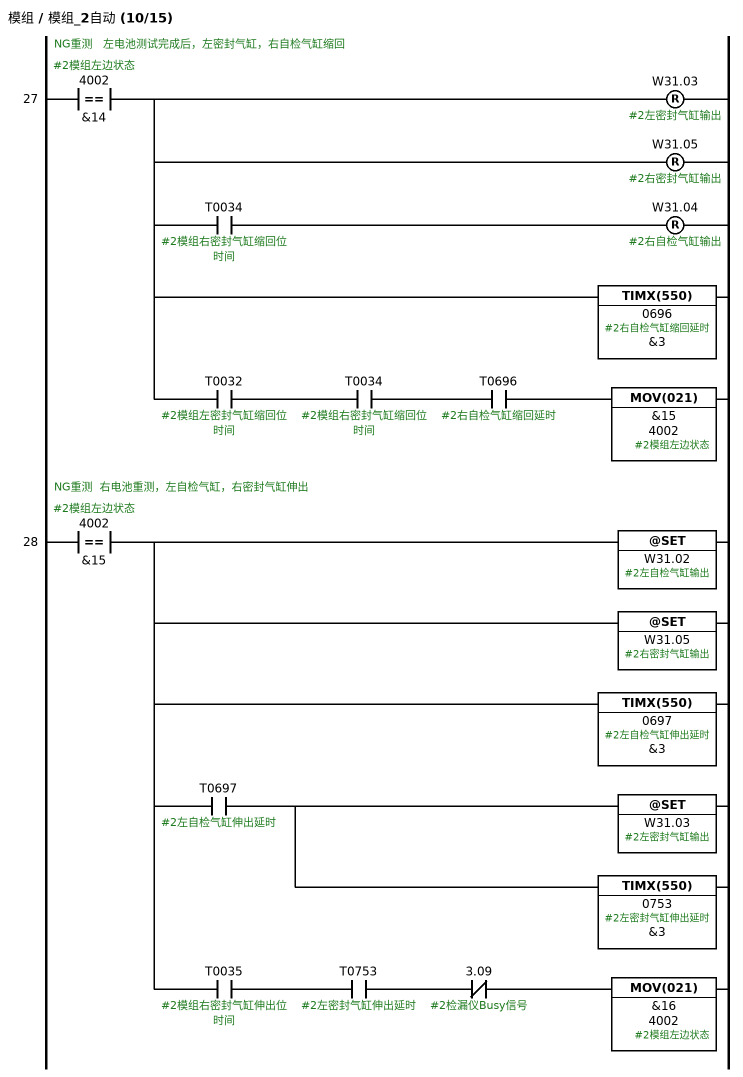
; rung 27: NG重测   左电池测试完成后，左密封气缸，右自检气缸缩回
LD=(300) 4002 &14  ; #2模组左边状态
OUT TR0
RSET W31.03  ; #2左密封气缸输出
RSET W31.05  ; #2右密封气缸输出
AND T0034  ; #2模组右密封气缸缩回位时间
RSET W31.04  ; #2右自检气缸输出
LD TR0
TIMX(550) 0696 &3  ; #2右自检气缸缩回延时
AND T0032  ; #2模组左密封气缸缩回位时间
AND T0034  ; #2模组右密封气缸缩回位时间
AND T0696  ; #2右自检气缸缩回延时
MOV(021) &15 4002  ; #2模组左边状态
; rung 28: NG重测  右电池重测，左自检气缸，右密封气缸伸出
LD=(300) 4002 &15  ; #2模组左边状态
OUT TR0
@SET W31.02  ; #2左自检气缸输出
@SET W31.05  ; #2右密封气缸输出
TIMX(550) 0697 &3  ; #2左自检气缸伸出延时
AND T0697  ; #2左自检气缸伸出延时
@SET W31.03  ; #2左密封气缸输出
TIMX(550) 0753 &3  ; #2左密封气缸伸出延时
LD TR0
AND T0035  ; #2模组右密封气缸伸出位时间
AND T0753  ; #2左密封气缸伸出延时
ANDNOT 3.09  ; #2检漏仪Busy信号
MOV(021) &16 4002  ; #2模组左边状态

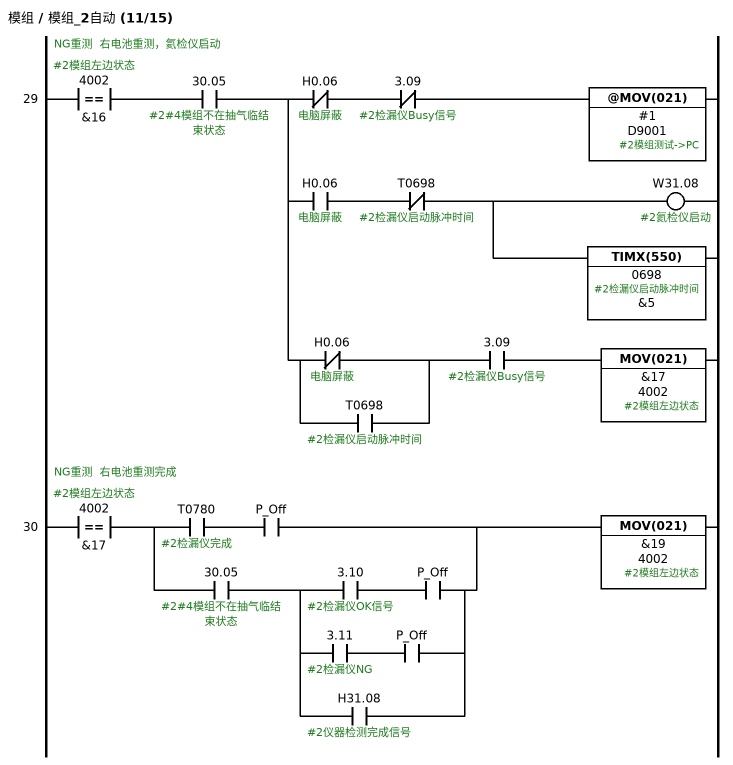
; rung 29: NG重测  右电池重测，氦检仪启动
LD=(300) 4002 &16  ; #2模组左边状态
AND 30.05  ; #2#4模组不在抽气临结束状态  // 2018/5/28hy修改 所有模组不在抽气临结束状态下，下一模组才能启动(防抽气NG)
OUT TR0
ANDNOT H0.06  ; 电脑屏蔽
ANDNOT 3.09  ; #2检漏仪Busy信号
@MOV(021) #1 D9001  ; #2模组测试->PC
LD TR0
AND H0.06  ; 电脑屏蔽
ANDNOT T0698  ; #2检漏仪启动脉冲时间
OUT W31.08  ; #2氦检仪启动
TIMX(550) 0698 &5  ; #2检漏仪启动脉冲时间
LD TR0
LDNOT H0.06  ; 电脑屏蔽
OR T0698  ; #2检漏仪启动脉冲时间
ANDLD
AND 3.09  ; #2检漏仪Busy信号
MOV(021) &17 4002  ; #2模组左边状态
; rung 30: NG重测  右电池重测完成
LD=(300) 4002 &17  ; #2模组左边状态
LD T0780  ; #2检漏仪完成
AND P_Off
LD 30.05  ; #2#4模组不在抽气临结束状态  // 2018/5/29hy修改,所有模组不在临抽气结束状态下，测试模组测试完成后，给出停止测试信号
LD 3.10  ; #2检漏仪OK信号
AND P_Off
LD 3.11  ; #2检漏仪NG
AND P_Off
ORLD
OR H31.08  ; #2仪器检测完成信号
ANDLD
ORLD
ANDLD
MOV(021) &19 4002  ; #2模组左边状态

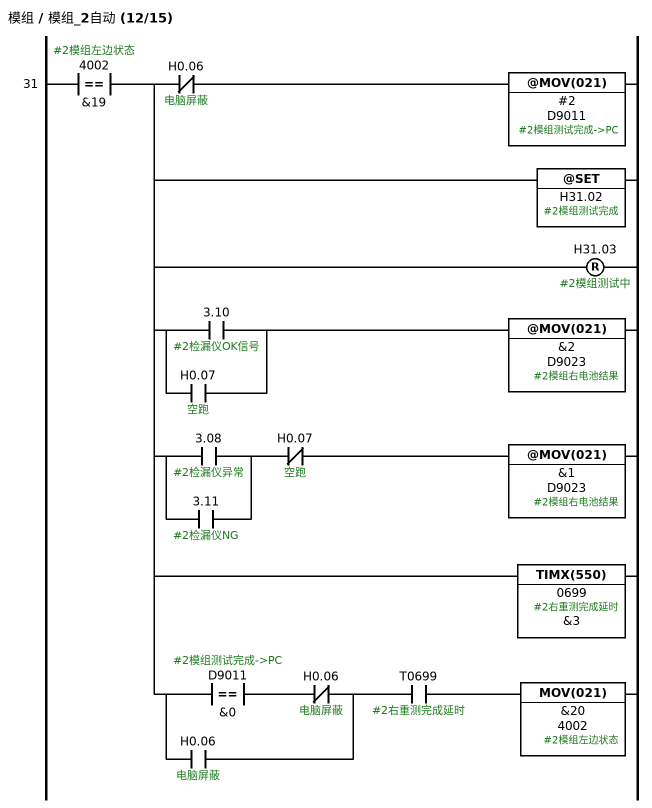
; rung 31
LD=(300) 4002 &19  ; #2模组左边状态
OUT TR0
ANDNOT H0.06  ; 电脑屏蔽
@MOV(021) #2 D9011  ; #2模组测试完成->PC
LD TR0
@SET H31.02  ; #2模组测试完成
RSET H31.03  ; #2模组测试中
LD 3.10  ; #2检漏仪OK信号
OR H0.07  ; 空跑
ANDLD
@MOV(021) &2 D9023  ; #2模组右电池结果
LD TR0
LD 3.08  ; #2检漏仪异常
OR 3.11  ; #2检漏仪NG
ANDLD
ANDNOT H0.07  ; 空跑
@MOV(021) &1 D9023  ; #2模组右电池结果
LD TR0
TIMX(550) 0699 &3  ; #2右重测完成延时
LD=(300) D9011 &0  ; #2模组测试完成->PC
ANDNOT H0.06  ; 电脑屏蔽
OR H0.06  ; 电脑屏蔽
ANDLD
AND T0699  ; #2右重测完成延时
MOV(021) &20 4002  ; #2模组左边状态

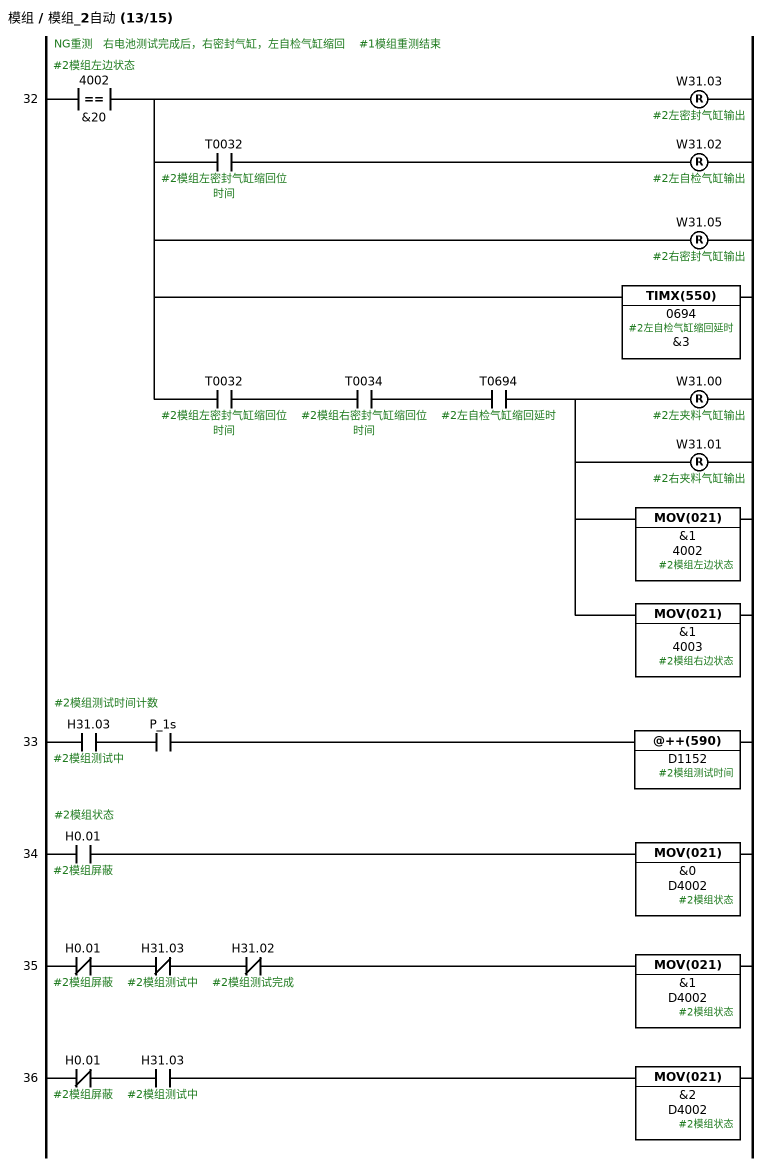
; rung 32: NG重测   右电池测试完成后，右密封气缸，左自检气缸缩回    #1模组重测结束
LD=(300) 4002 &20  ; #2模组左边状态
OUT TR0
RSET W31.03  ; #2左密封气缸输出
AND T0032  ; #2模组左密封气缸缩回位时间
RSET W31.02  ; #2左自检气缸输出
LD TR0
RSET W31.05  ; #2右密封气缸输出
TIMX(550) 0694 &3  ; #2左自检气缸缩回延时
AND T0032  ; #2模组左密封气缸缩回位时间
AND T0034  ; #2模组右密封气缸缩回位时间
AND T0694  ; #2左自检气缸缩回延时
RSET W31.00  ; #2左夹料气缸输出
RSET W31.01  ; #2右夹料气缸输出
MOV(021) &1 4002  ; #2模组左边状态
MOV(021) &1 4003  ; #2模组右边状态
; rung 33: #2模组测试时间计数
LD H31.03  ; #2模组测试中
AND P_1s
@++(590) D1152  ; #2模组测试时间
; rung 34: #2模组状态
LD H0.01  ; #2模组屏蔽
MOV(021) &0 D4002  ; #2模组状态
; rung 35
LDNOT H0.01  ; #2模组屏蔽
ANDNOT H31.03  ; #2模组测试中
ANDNOT H31.02  ; #2模组测试完成
MOV(021) &1 D4002  ; #2模组状态
; rung 36
LDNOT H0.01  ; #2模组屏蔽
AND H31.03  ; #2模组测试中
MOV(021) &2 D4002  ; #2模组状态

